{attribute 'qualified_only'}
VAR_GLOBAL
		myInt1:INT;
END_VAR

(* stored: Version 1.1.0.1, ProductVersion 3.1.4022.18
   GVL GVL_1: Id {9634ded6-8da4-41a3-805d-c800cc5fd4b3} *)
